{attribute 'qualified_only'}
{attribute 'conditionalshow'}
VAR_GLOBAL	
	refSystem 			: REFERENCE TO FB_System;		
END_VAR

(* stored: Version 1.1.0.1, ProductVersion 3.1.4024.13
   GVL GVL_Core: Id {daaa4602-82dd-0eaa-0bd4-a2e6b9fa282a}
   Property fbSystem: Id {d875db5b-3f7e-02b0-230c-ed0ec43a556a}
   Get Get: Id {b76067e0-6c2d-0f93-3724-711b1b967692} *)
